// TIA Portal V17 export
// export: Created 2022-06-27T14:01:00.8233571Z, ExportSetting WithDefaults, DisplayName Totally Integrated Automation Portal, DisplayVersion V17 Update 3, DisplayName TIA Portal Openness, DisplayVersion V17 Update 3, DisplayName TIA Portal Version Control Interface, DisplayVersion V17, DisplayName SINAMICS Startdrive Advanced, DisplayVersion V17 Update1, DisplayName SINAMICS Startdrive G110M, G120, G120C, G120D, G120P, G115D, DisplayVersion V17 Update1, DisplayName SINAMICS Startdrive G130, G150, S120, S150, SINAMICS MV, S210, DisplayVersion V17 Update1, DisplayName STEP 7 Professional, DisplayVersion V17 Update 3, DisplayName STEP 7 Safety, DisplayVersion V17, DisplayName WinCC UA Professional, DisplayVersion V17 Update 3
VAR_GLOBAL   // PLC tag table "A6-9F"
   "LSL66-2C" AT %I40.0 : Bool;   // Sensor de nível do catador
   "A66-2E_I40-0" AT %I40.1 : Bool;   // Reserva I40.0
   "ZSL66-4B" AT %I40.2 : Bool;   // Fim de curso alimenta câmara 1 - fechado
   "ZSH66-5B" AT %I40.3 : Bool;   // Fim de curso alimenta câmara 1 - aberto
   "ZSL66-6B" AT %I40.4 : Bool;   // Fim de curso descarga câmara 1 - fechado
   "ZSH66-7B" AT %I40.5 : Bool;   // Fim de curso descarga câmara 1 - aberto
   "ZSL66-8B" AT %I40.6 : Bool;   // Fim de curso descarga esfriador 1 - fechado
   "ZSH66-9B" AT %I40.7 : Bool;   // Fim de curso descarga esfriador 1 - aberto
   "ZSL67-2B" AT %I41.0 : Bool;   // Fim de curso alimenta câmara 2 - fechado
   "ZSH67-3B" AT %I41.1 : Bool;   // Fim de curso alimenta câmara 2 - aberto
   "ZSL67-4B" AT %I41.2 : Bool;   // Fim de curso descarga câmara 2 - fechado
   "ZSH67-5B" AT %I41.3 : Bool;   // Fim de curso descarga câmara 2 - aberto
   "ZSL67-6B" AT %I41.4 : Bool;   // Fim de curso descarga esfriador 2 - fechado
   "ZSH67-7B" AT %I41.5 : Bool;   // Fim de curso descarga esfriador 2 - aberto
   "ZSL67-8B" AT %I41.6 : Bool;   // Fim de curso ventilador torrando câmara 2
   "ZSH67-9B" AT %I41.7 : Bool;   // Fim de curso ventilador torrando câmara 1
   "ZSL68-2B" AT %I42.0 : Bool;   // Fim de curso ventilador secando câmara 2
   "ZSH68-3B" AT %I42.1 : Bool;   // Fim de curso ventilador secando câmara 1
   "ZSL68-4B" AT %I42.2 : Bool;   // Fim de curso ventilador esfriando câmara 1
   "ZSH68-5B" AT %I42.3 : Bool;   // Fim de curso ventilador esfriando câmara 2
   "ZSL68-6B" AT %I42.4 : Bool;   // Registro derivador sentido ensaque manual
   "ZSH68-7B" AT %I42.5 : Bool;   // Registro derivador sentido transporte
   "ZSL68-8B" AT %I42.6 : Bool;   // Registro derivador de transporte sentido elevador
   "ZSH68-9B" AT %I42.7 : Bool;   // Registro derivador de transporte sentido catador
   "LSH69-2B" AT %I43.0 : Bool;   // Sensor capacitivo silo café cru câmara 1 nível 1
   "LSL69-3B" AT %I43.1 : Bool;   // Sensor capacitivo silo café cru câmara 1 nível 2
   "A68-2E_I43-2" AT %I43.2 : Bool;   // Reserva I43.2
   "LSH69-5B" AT %I43.3 : Bool;   // Sensor capacitivo silo café cru câmara 2 nível 1
   "LSL69-6B" AT %I43.4 : Bool;   // Sensor capacitivo silo café cru câmara 2 nível 2
   "A68-2E_-43-5" AT %I43.5 : Bool;   // Reserva I43.5
   "SSL69-8B" AT %I43.6 : Bool;   // Sensor de giro eixo com pás câmara 1
   "SSL69-9B" AT %I43.7 : Bool;   // Sensor de giro eixo com pás câmara 2
   "SSL70-2B" AT %I44.0 : Bool;   // Sensor de giro eixo com pás esfriador 1
   "SSL70-3B" AT %I44.1 : Bool;   // Sensor de giro eixo com pás esfriador 2
   "SSL70-4B" AT %I44.2 : Bool;   // Sensor de giro rosca sob esfriador
   "SSL70-5B" AT %I44.3 : Bool;   // Sensor de giro rosca inclinada
   "LSL70-6B" AT %I44.4 : Bool;   // Sensor nível tanque de água
   "LSL70-7B" AT %I44.5 : Bool;   // Sensor capacitivo caçamba esfriador 1
   "LSL70-8B" AT %I44.6 : Bool;   // Sensor capacitivo caçamba esfriador 2
   "PSL70-9B" AT %I44.7 : Bool;   // Pressostato ar comprimido
   "HR71-2BA" AT %I45.0 : Bool;   // Válvula manual alimenta bomba de água - aberta
   "HR71-2BF" AT %I45.1 : Bool;   // Válvula manual alimenta bomba de água - fechada
   "ZSL71-4B" AT %I45.2 : Bool;   // Micro final rosca sob ciclones
   "ZSL71-5B" AT %I45.3 : Bool;   // Micro final rosca inclinada
   "ZSH71-5B" AT %I45.4 : Bool;   // Atuador pneumático ar quente câmara 1 - aberto
   "ZSL71-7B" AT %I45.5 : Bool;   // Atuador pneumático ar quente câmara 1 - fechado
   "ZSH71-8B" AT %I45.6 : Bool;   // Atuador pneumático ar quente câmara 2 - aberto
   "ZSL71-9B" AT %I45.7 : Bool;   // Atuador pneumático ar quente câmara 2 - fechado
   "ZSH72-2B" AT %I46.0 : Bool;   // Atuador pneumático ar ambiente câmara 1 - aberto
   "ZSL72-3B" AT %I46.1 : Bool;   // Atuador pneumático ar ambiente câmara 1 - fechado
   "ZSH72-4B" AT %I46.2 : Bool;   // Atuador pneumático ar ambiente câmara 2 - aberto
   "ZSL72-5B" AT %I46.3 : Bool;   // Atuador pneumático ar ambiente câmara 2 - fechado
   "SSL72-6B" AT %I46.4 : Bool;   // Sensor de giro válvula rotativa ciclone torrador
   "SSL72-7B" AT %I46.5 : Bool;   // Sensor de giro ventilador torrador
   "SSL72-8B" AT %I46.6 : Bool;   // Sensor de giro ventilador secador
   "PSL72-9B" AT %I46.7 : Bool;   // Sensor de giro ventilador esfriador
   "S73-2B" AT %I47.0 : Bool;   // Chave de ensaque em manual
   "S73-3B" AT %I47.1 : Bool;   // Chave de ensaque em automático
   "PSL73-4B" AT %I47.2 : Bool;   // Pressostato ventilador ar ambiente câmara 1
   "PSL73-5B" AT %I47.3 : Bool;   // Pressostato ventilador ar ambiente câmara 2
   "SSL73-6B" AT %I47.4 : Bool;   // Sensor de giro válvula rotativa ciclone esfriador
   "SSL73-7B" AT %I47.5 : Bool;   // Sensor de giro válvula rotativa ciclone 1 secador
   "SSL73-8B" AT %I47.6 : Bool;   // Sensor de giro válvula rotativa ciclone 2 secador
   "SSL73-9B" AT %I47.7 : Bool;   // Sensor de giro rosca sob ciclones
   "HSH74-2B" AT %I48.0 : Bool;   // Válvula manual alimentaçâo de ar aberta
   "HSL74-3B" AT %I48.1 : Bool;   // Válvula manual de injeçâo de água câmara 1 - fechado
   "HSL74-4B" AT %I48.2 : Bool;   // Válvula manual de injeçâo de água câmara 2 - fechado
   "HSL74-5B" AT %I48.3 : Bool;   // Válvula manual de injeçâo de água esfriador 1 - fechado
   "HSL74-6B" AT %I48.4 : Bool;   // Válvula manual de injeçâo de água esfriador 2 - fechado
   "HSL74-7B" AT %I48.5 : Bool;   // Válvula manual alívio tanque de ar - fechado
   "HSL74-8B" AT %I48.6 : Bool;   // Válvula manual alívio ar tanque de água - fechado
   "HSH74-9B" AT %I48.7 : Bool;   // Válvula manual alimenta torrador após bomba de água - aberta
   "HSH75-2B" AT %I49.0 : Bool;   // Válvula manual alimenta água para torrador - aberta
   "HSH75-3B" AT %I49.1 : Bool;   // Válvula manual água de aromatização - aberta
   "PSL75-4B" AT %I49.2 : Bool;   // Pressostato medição de entrada de ar
   "FSL75-5B" AT %I49.3 : Bool;   // Medição vazão de água
   "ZSL75-6B" AT %I49.4 : Bool;   // Fim de curso rosca sob esfriador
   "K94-4D" AT %I49.5 : Bool;   // Medição vazão de gás
   "K94-7D" AT %I49.6 : Bool;   // Medição vazão de óleo
   "A74-2E_I49-7" AT %I49.7 : Bool;   // Reserva I49.7
   "HSV76-2B" AT %I50.0 : Bool;   // Reserva I50.0
   "HSV76-3B" AT %I50.1 : Bool;   // Reserva I50.1
   "HSV76-4B" AT %I50.2 : Bool;   // Reserva I50.2
   "HSV76-5B" AT %I50.3 : Bool;   // Reserva I50.3
   "A76-2E_I50-4" AT %I50.4 : Bool;   // Reserva I50.4
   "A76-2E_I50-5" AT %I50.5 : Bool;   // Reserva I50.5
   "A76-2E_I50-6" AT %I50.6 : Bool;   // Reserva I50.6
   "A76-2E_I50-7" AT %I50.7 : Bool;   // Reserva I50.7
   "A76-2E_I51-0" AT %I51.0 : Bool;   // Reserva I51.0
   "A76-2E_I51-1" AT %I51.1 : Bool;   // Reserva I51.1
   "A76-2E_I51-2" AT %I51.2 : Bool;   // Reserva I51.2
   "A76-2E_I51-3" AT %I51.3 : Bool;   // Reserva I51.3
   "A76-2E_I51-4" AT %I51.4 : Bool;   // Reserva I51.4
   "A76-2E_I51-5" AT %I51.5 : Bool;   // Reserva I51.5
   "A76-2E_I51-6" AT %I51.6 : Bool;   // Reserva I51.6
   "A76-2E_I51-7" AT %I51.7 : Bool;   // Reserva I51.7
   "FV78-2E" AT %Q16.0 : Bool;   // Limpeza cano de água câmara 1
   "FV78-3E" AT %Q16.1 : Bool;   // Limpeza cano de água câmara 2
   "FV78-4E" AT %Q16.2 : Bool;   // Tanque pressurização
   "K92-6E" AT %Q16.3 : Bool;   // Auxiliar aromatização câmara 1
   "FV78-6E" AT %Q16.4 : Bool;   // Emergência incêndio esfriador 1
   "K92-7E" AT %Q16.5 : Bool;   // Auxiliar aromatização câmara 2
   "FV78-8E" AT %Q16.6 : Bool;   // Emergência incêndio esfriador 2
   "FV78-9E" AT %Q16.7 : Bool;   // Solenoide água rosca de películas
   "FV79-2E" AT %Q17.0 : Bool;   // Alívio tanque de água
   "FV79-3E" AT %Q17.1 : Bool;   // Alimenta tanque de água
   "FV79-4E" AT %Q17.2 : Bool;   // Solenoide água emergência rosca de películas
   "A78-2E_Q17-3" AT %Q17.3 : Bool;   // Reserva Q17.3
   "A78-2E_Q17-4" AT %Q17.4 : Bool;   // Reserva Q17.4
   "A78-2E_Q17-5" AT %Q17.5 : Bool;   // Reserva Q17.5
   "A78-2E_Q17-6" AT %Q17.6 : Bool;   // Reserva Q17.6
   "A78-2E_Q17-7" AT %Q17.7 : Bool;   // Reserva Q17.7
   "A80-2B_Q18-0" AT %Q18.0 : Bool;   // Reserva Q18.0
   "A80-2B_Q18-1" AT %Q18.1 : Bool;   // Reserva Q18.1
   "A80-2B_Q18-2" AT %Q18.2 : Bool;   // Reserva Q18.2
   "A80-2B_Q18-3" AT %Q18.3 : Bool;   // Reserva Q18.3
   "A80-2B_Q18-4" AT %Q18.4 : Bool;   // Reserva Q18.4
   "A80-2B_Q18-5" AT %Q18.5 : Bool;   // Reserva Q18.5
   "A80-2B_Q18-6" AT %Q18.6 : Bool;   // Reserva Q18.6
   "A80-2B_Q18-7" AT %Q18.7 : Bool;   // Reserva Q18.7
   "A80-2B_Q19-0" AT %Q19.0 : Bool;   // Reserva Q19.0
   "A80-2B_Q19-1" AT %Q19.1 : Bool;   // Reserva Q19.1
   "A80-2B_Q19-2" AT %Q19.2 : Bool;   // Reserva Q19.2
   "A80-2B_Q19-3" AT %Q19.3 : Bool;   // Reserva Q19.3
   "A80-2B_Q19-4" AT %Q19.4 : Bool;   // Reserva Q19.4
   "A80-2B_Q19-5" AT %Q19.5 : Bool;   // Reserva Q19.5
   "A80-2B_Q19-6" AT %Q19.6 : Bool;   // Reserva Q19.6
   "A80-2B_Q19-7" AT %Q19.7 : Bool;   // Reserva Q19.7
   "TT82-2E" AT %IW52 : Int;   // Temperatura fornalha
   "TT82-4E" AT %IW54 : Int;   // Temperatura entrada de ar câmara 1
   "TT82-6E" AT %IW56 : Int;   // Temperatura entrada de ar câmara 2
   "TT82-8E" AT %IW58 : Int;   // Temperatura de retorno
   "TT83-2E" AT %IW60 : Int;   // Temperatura 1 ciclone torrando
   "A83-2E_IW62" AT %IW62 : Int;   // Reserva IW62
   "TT83-6E" AT %IW64 : Int;   // Temperatura 1 câmara 1
   "TT83-8E" AT %IW66 : Int;   // Temperatura 1 câmara 2
   "TT84-2E" AT %IW68 : Int;   // Temperatura 2 câmara 1
   "TT84-4E" AT %IW70 : Int;   // Temperatura 2 câmara 2
   "TT84-6E" AT %IW72 : Int;   // Temperatura esfriador 1
   "TT84-8E" AT %IW74 : Int;   // Temperatura esfriador 2
   "TT85-2E" AT %IW76 : Int;   // Temperatura queima de fumaça fornalha
   "TT85-4E" AT %IW78 : Int;   // Temperatura rosca de películas
   "A85-2E_IW80" AT %IW80 : Int;   // Reserva IW80
   "A85-2E_IW82" AT %IW82 : Int;   // Reserva IW82
   "FY86-2E" AT %QW20 : Int;   // Comando posicionador pneumático ar quente câmara 1
   "FY86-4E" AT %QW22 : Int;   // Comando posicionador pneumático ar ambiente câmara 1
   "FY86-6E" AT %QW24 : Int;   // Comando posicionador pneumático ar quente câmara 2
   "FY86-8E" AT %QW26 : Int;   // Comando posicionador pneumático ar ambiente câmara 2
   "VR87-2E" AT %IW84 : Int;   // Sensor vibração mancal traseiro ventilador torrando
   "VR87-4E" AT %IW86 : Int;   // Sensor vibração mancal dianteiro ventilador torrando
   "VR87-6E" AT %IW88 : Int;   // Sensor vibração mancal traseiro ventilador secando
   "VR87-8E" AT %IW90 : Int;   // Sensor vibração mancal dianteiro ventilador secando
   "A87-2B_IW92" AT %IW92 : Int;   // Reserva IW92
   "A87-2B_IW94" AT %IW94 : Int;   // Reserva IW94
   "A87-2B_IW96" AT %IW96 : Int;   // Reserva IW96
   "A87-2B_IW98" AT %IW98 : Int;   // Reserva IW98
   "BCV98-2B" AT %IW100 : Int;   // Sinal setpoint velocidade queimador
   "A89-2B_IW102" AT %IW102 : Int;   // Reserva IW102
   "A89-2B_IW104" AT %IW104 : Int;   // Reserva IW104
   "A89-2B_IW106" AT %IW106 : Int;   // Reserva IW106
   "A89-2B_IW108" AT %IW108 : Int;   // Reserva IW108
   "A89-2B_IW110" AT %IW110 : Int;   // Reserva IW110
   "A89-2B_IW112" AT %IW112 : Int;   // Reserva IW112
   "A89-2B_IW114" AT %IW114 : Int;   // Reserva IW114
   "BCV98F-2B" AT %QW28 : Int;   // Regulador de potência queimador
   "A90-2B_QW30" AT %QW30 : Int;   // Reserva QW30
   "A90-2B_QW32" AT %QW32 : Int;   // Reserva QW32
   "A90-2B_QW34" AT %QW34 : Int;   // Reserva QW34
END_VAR
